TYPE ST_AutoMode_DetectDiameter :
STRUCT
	Command: ST_DetectDiameterCommand;
	Status: ST_DetectDiameterStatus;
	DetectDiameterInfo:ST_DetectDiameterInfo;
END_STRUCT
END_TYPE

(* stored: Version 1.1.0.1, ProductVersion 3.1.4024.13
   DUT ST_AutoMode_DetectDiameter: Id {0ae85748-950a-48cd-9285-a6b5eab03c78} *)
